(* PLC project Unnamed, Unknown Unnamed 1 *)
(* stored: creationDateTime 2025-12-31T15:27:39, modificationDateTime 2025-12-31T15:27:39 *)

PROGRAM main
  VAR
    SW1 AT %IX0.3 : BOOL;
    SW2 AT %IX0.4 : BOOL;
    CR1 AT %QX2.0 : BOOL;
    CR2 AT %QX2.1 : BOOL;
    CR3 AT %QX0.0 : BOOL;
  END_VAR
  VAR
    CR : BOOL;
    CR4 : BOOL;
    CR5 : BOOL;
    CR6 : BOOL;
    CR7 : BOOL;
  END_VAR

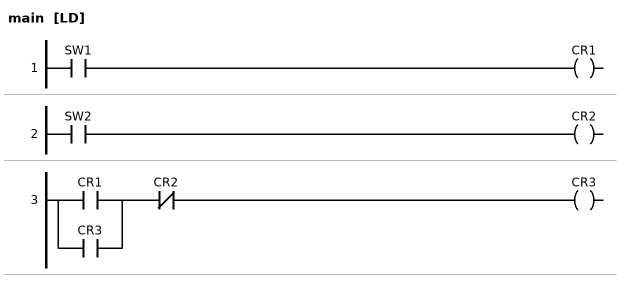
(* LD diagram, written out as Structured Text *)
CR1 := SW1;
CR2 := SW2;
CR3 := (CR1 OR CR3) AND NOT CR2;
END_PROGRAM

CONFIGURATION Config0
  RESOURCE Res0 ON PLC
    TASK task0(INTERVAL := T#20ms, PRIORITY := 1);
    PROGRAM instance0 WITH task0 : main;
  END_RESOURCE
END_CONFIGURATION
